// TIA Portal V19 export
FUNCTION "F11_PLC1" : Void   // FC112, STL
TITLE = IF 1 Wort ohne Bit Signale
{ S7_Optimized_Access := 'TRUE' }
AUTHOR : RFu
FAMILY : PLC
NAME : PLC1
// stored: AutoNumber false
   VAR_INPUT
      IW_PS : Word;   // Eingang Prozesssignal
      IR_Gradient : Real;   // Gradient
   END_VAR
   VAR_OUTPUT
      OR_PS : Real;   // Ausgabe Prozesssignal
   END_VAR
BEGIN

NETWORK
TITLE = 
// Prozesssignal 1
      L     #IR_Gradient;
      L     0.0;
      ==R;
      JCN   xxxx;
      L     1.0;
      T     #IR_Gradient;
xxxx: NOP   0;

      L     #IW_PS;
      ITD;
      DTR;
      L     #IR_Gradient;
      *R;
      T     #OR_PS;






END_FUNCTION
